TYPE ST_Ifm_TX :
STRUCT
	InputByte : ARRAY[0..3] OF USINT;
END_STRUCT
END_TYPE

(* stored: Version 1.1.0.1, ProductVersion 3.1.4024.12
   DUT ST_Ifm_TX: Id {67e96d0f-8190-44b3-8b95-2fbdfbc010c7} *)
